FUNCTION_BLOCK FB_SYSTEM_SeqControl
VAR_INPUT
	nSeqStepNo	: INT;
END_VAR
VAR_OUTPUT
	bActive		: BOOL;
	bStep00		: BOOL;
	bStep01		: BOOL;
	bStep02		: BOOL;
	bStep03		: BOOL;
	bStep04		: BOOL;
	bStep05		: BOOL;
	bStep06		: BOOL;
	bStep07		: BOOL;
	bStep08		: BOOL;
	bStep09		: BOOL;
	bStep10		: BOOL;
	bStep11		: BOOL;
	bStep12		: BOOL;
	bStep13		: BOOL;
	bStep14		: BOOL;
	bStep15		: BOOL;
	bStep16		: BOOL;
	bStep17		: BOOL;
	bStep18		: BOOL;
	bStep19		: BOOL;
	bStep20		: BOOL;
END_VAR
VAR
END_VAR
(*
-------------------------------------------------------------------------------------------------
Date		Version	Author	Comments
-------------------------------------------------------------------------------------------------
30/01/2015	3.00.00	PB		Initial release

-------------------------------------------------------------------------------------------------
*)

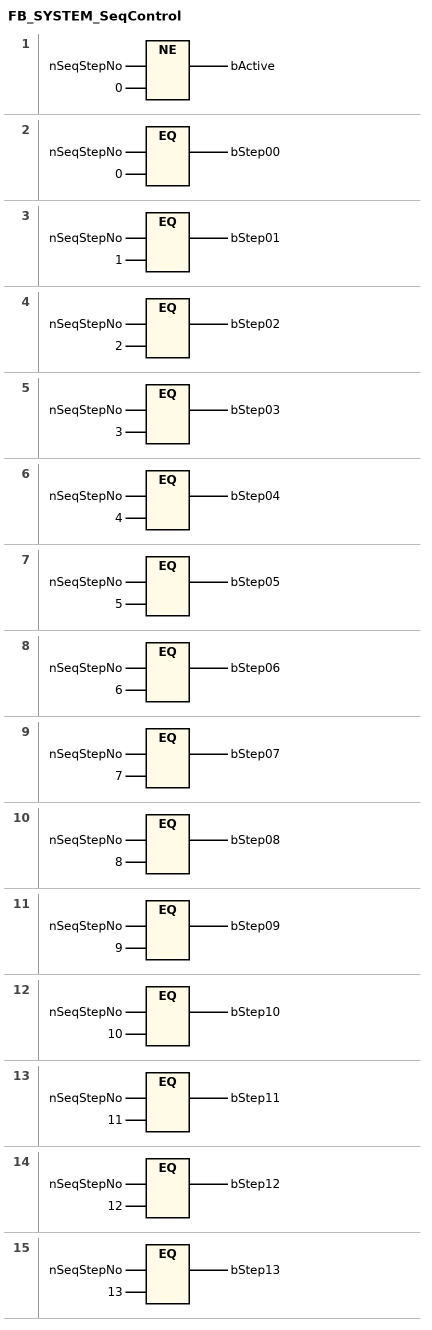
// NETWORK 1
bActive := nSeqStepNo <> 0;

// NETWORK 2
bStep00 := nSeqStepNo = 0;

// NETWORK 3
bStep01 := nSeqStepNo = 1;

// NETWORK 4
bStep02 := nSeqStepNo = 2;

// NETWORK 5
bStep03 := nSeqStepNo = 3;

// NETWORK 6
bStep04 := nSeqStepNo = 4;

// NETWORK 7
bStep05 := nSeqStepNo = 5;

// NETWORK 8
bStep06 := nSeqStepNo = 6;

// NETWORK 9
bStep07 := nSeqStepNo = 7;

// NETWORK 10
bStep08 := nSeqStepNo = 8;

// NETWORK 11
bStep09 := nSeqStepNo = 9;

// NETWORK 12
bStep10 := nSeqStepNo = 10;

// NETWORK 13
bStep11 := nSeqStepNo = 11;

// NETWORK 14
bStep12 := nSeqStepNo = 12;

// NETWORK 15
bStep13 := nSeqStepNo = 13;

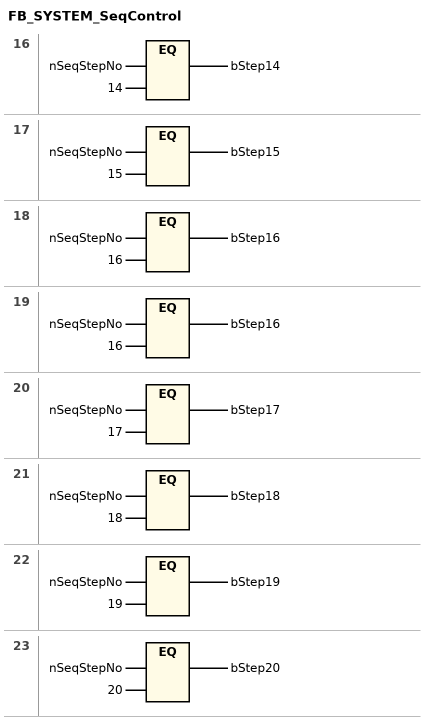
// NETWORK 16
bStep14 := nSeqStepNo = 14;

// NETWORK 17
bStep15 := nSeqStepNo = 15;

// NETWORK 18
bStep16 := nSeqStepNo = 16;

// NETWORK 19
bStep16 := nSeqStepNo = 16;

// NETWORK 20
bStep17 := nSeqStepNo = 17;

// NETWORK 21
bStep18 := nSeqStepNo = 18;

// NETWORK 22
bStep19 := nSeqStepNo = 19;

// NETWORK 23
bStep20 := nSeqStepNo = 20;

END_FUNCTION_BLOCK

(* stored: Version 1.1.0.1
   POU FB_SYSTEM_SeqControl: Id {c6a1f4f7-49a9-4048-bd3e-a0801da15808}, SpecialFunc None *)
